(* IEC 61131-3 sources: paho.mqtt.c-ar/Samples/IotMqttSamples/SampleTasks/AWSIoT, 3 files *)

(* ---- Main.st ---- *)
PROGRAM _CYCLIC

	Parameters;

	IotMqttClient_0.Enable			:= TRUE;
	IotMqttClient_0.Connect			:= TRUE;
	IotMqttClient_0.IotMqttLink 	:= ADR(IotMqttLink);
	IotMqttClient_0.Parameters		:= IotMqttParameters;
	IotMqttClient_0();

	PublishTopic	:= 'B&R/Telemetry';	//Could be any topic
	SubscribeTopic	:= 'B&R/Receive';	//Could be any topic
	brsstrcat(ADR(PublishTopic),ADR(ClientID));

	Publish;
	Subscribe;

END_PROGRAM

PROGRAM _EXIT

    IotMqttClient_0(Enable	:= FALSE);
    IotMqttPublish_0(Enable	:= FALSE);
    IotMqttSubscribe_0(Enable := FALSE);

END_PROGRAM

(* ---- Parameters.st ---- *)
ACTION Parameters:

	IotMqttParameters.ConnectionType			:= IotMqtt_TCP;
	IotMqttParameters.ClientID					:= 'BR_CoffeeMachine';
	IotMqttParameters.ServerUri					:= 'Must be filled with your device endpoint, obtained at the AWS IoT portal';
	IotMqttParameters.Port						:= 8883;
	IotMqttParameters.CleanSession				:= FALSE;
	IotMqttParameters.KeepAliveInterval			:= T#30s;
	IotMqttParameters.AutomaticReconnect		:= TRUE;

	IotMqttParameters.TLS.UseTLS				:= TRUE;
	IotMqttParameters.TLS.CA					:= ADR('//CS:EXT/AmazonRootCA1.pem');
	IotMqttParameters.TLS.Cert					:= ADR('//CS:OWN/BR_CoffeeMachine_certificate.pem.crt'); //Aws thing certificate, downloaded from Aws Iot portal
	IotMqttParameters.TLS.PrivateKey			:= ADR('//CS:KEY/BR_CoffeeMachine_private.pem.key');//Aws thing private key, downloaded from Aws Iot portal
	IotMqttParameters.TLS.EnableServerCertAuth	:= TRUE;

END_ACTION

(* ---- Subscribe.st ---- *)
ACTION Subscribe:

	IotMqttSubscribe_0.Enable := TRUE;
	IotMqttSubscribe_0.IotMqttLink			:= IotMqttClient_0.IotMqttLink;
	IotMqttSubscribe_0.Topic				:= ADR(SubscribeTopic);
	IotMqttSubscribe_0.SubscriptionQoS		:= IotMqtt_QoS1;
	IotMqttSubscribe_0.RecievedTopic		:= ADR(ReceivedTopic);
	IotMqttSubscribe_0.RecievedTopicSize	:= SIZEOF(ReceivedTopic);
	IotMqttSubscribe_0.QueueSize 			:= 50;
	IotMqttSubscribe_0.Buffer				:= ADR(ReceiveBuffer);
	IotMqttSubscribe_0.BufferSize	 		:= SIZEOF(ReceiveBuffer);
	IotMqttSubscribe_0();

END_ACTION
